FUNCTION_BLOCK FB_Analog
VAR_INPUT
END_VAR
VAR_OUTPUT
END_VAR
VAR
END_VAR

//***********************************************************************************
//
// ETH Zürich / Robotic Fabrication Lab
// HIB C 13 / Stefano-Franscini-Platz 1
// CH-8093 Zürich
// 
// ***********************************************************************************
// 
// PROJECT     :  ?? 
// 
// FUNCTION    :  Analog Calculation
// 
// AUTHOR      :  Mathias Suter
// 
// EMAIL       :  mathias.suter@solinaut.ch
// 
// Copyright   :  ETH Zürich (CH) 2021
//
// ***********************************************************************************


//
// Analog Inputs - Scale 0-100%
GVL.fControlMixerPumpSpeed := INT_TO_REAL(GVL.nControlMixerPumpSpeed) / 32767 * 100;			
//GVL.fControlPeristalticPumpSpeed := INT_TO_REAL(GVL.nControlPeristalticPumpSpeed) / 32767 * 100;			
GVL.fControlDosingPumpSpeed := INT_TO_REAL(GVL.nControlDosingPumpSpeed) / 32767 * 100;				
GVL.fInputSpare1 := INT_TO_REAL(GVL.nInputSpare1) / 32767 * 100;						
GVL.fInputSpare2 := INT_TO_REAL(GVL.nInputSpare2) / 32767 * 100;						
	

//
// Analog Outputs - Scale 0-100%
// GVL.nConcretePumpSpeed := REAL_TO_INT(GVL.fConcretePumpSpeed / 100 * 32767);				
GVL.nDosingPumpSpeed := REAL_TO_INT(GVL.fDosingPumpSpeed / 100 * 32767);					
GVL.nOutputSpare1 := REAL_TO_INT(GVL.fOutputSpare1 / 100 * 32767);						
GVL.nOutputSpare2 := REAL_TO_INT(GVL.fOutputSpare2 / 100 * 32767);

END_FUNCTION_BLOCK

(* stored: Version 1.1.0.1, ProductVersion 3.1.4024.11
   POU FB_Analog: Id {3c3a665e-cb0e-4117-b633-de110b8896f1}, SpecialFunc None *)
